Staubli VAL3: JointAccel.dtx

public num ja1
public num ja2
public num ja3
public num ja4
public num ja5
public num ja6
